{attribute 'GeneratedUsingTerminal: EL6201-0000-0017'}
{attribute addProperty BoxType "EL6201-0000-0017"}
{attribute addProperty Id "Slave_26A_DO0BOOL1Slave_26A_DO1BOOL1Slave_26A_DO2BOOL1Slave_26A_DO3BOOL1Slave_26B_DO0BOOL1Slave_26B_DO1BOOL1Slave_26B_DO2BOOL1Slave_26B_DO3BOOL1"}
{attribute addProperty CRC "2032404543"}
{attribute addProperty Size "8"}
TYPE Slave_26_Outputs_7924083F :
STRUCT
	{attribute addProperty Name "Slave_26A_DO0"}
	Slave_26A_DO0 : BOOL;
	{attribute addProperty Name "Slave_26A_DO1"}
	Slave_26A_DO1 : BOOL;
	{attribute addProperty Name "Slave_26A_DO2"}
	Slave_26A_DO2 : BOOL;
	{attribute addProperty Name "Slave_26A_DO3"}
	Slave_26A_DO3 : BOOL;
	{attribute addProperty Name "Slave_26B_DO0"}
	Slave_26B_DO0 : BOOL;
	{attribute addProperty Name "Slave_26B_DO1"}
	Slave_26B_DO1 : BOOL;
	{attribute addProperty Name "Slave_26B_DO2"}
	Slave_26B_DO2 : BOOL;
	{attribute addProperty Name "Slave_26B_DO3"}
	Slave_26B_DO3 : BOOL;
END_STRUCT
END_TYPE

(* stored: Version 1.2.0.0, ProductVersion 3.1.4024.11
   DUT Slave_26_Outputs_7924083F: Id {d35efe7a-02e8-4451-a752-37e8e2b66f00} *)
